{attribute 'linkalways'} 
{attribute 'no_explicit_call' := 'This FB is a CLASS and must be accessed using methods or properties'}
{attribute 'enable_dynamic_creation'}
FUNCTION_BLOCK Node_F_VN_HistogramExp EXTENDS VisionNode
VAR
	ipSrcImage : _ITcVnImage;
	ipMask : _ITcVnImage;
    ipDestHistogram : _ITcVnContainer;
	nBins : _UDINT(0);
	fLowerBound : _LREAL(0.0);
	fUpperBound : _LREAL(0.0);
    hrPrev : _HRESULT(S_OK);
	hresult : _HRESULT(S_OK);
END_VAR

METHOD PUBLIC  Clone : I_Node
VAR
	pNode : POINTER TO Node_F_VN_HistogramExp;
END_VAR
pNode := __NEW(Node_F_VN_HistogramExp);
Clone := pNode^;
END_METHOD

METHOD FB_init : BOOL
VAR_INPUT
	bInitRetains : BOOL; // if TRUE, the retain variables are initialized (warm start / cold start)
	bInCopyCode : BOOL;  // if TRUE, the instance afterwards gets moved into the copy code (online change)
END_VAR
AddInput('ipSrcImage', ipSrcImage);
AddInput('ipMask', ipMask);
AddInput('hrPrev', hrPrev);
AddParameter('nBins',nBins);
AddParameter('fLowerBound',fLowerBound);
AddParameter('fUpperBound',fUpperBound);
AddOutput('ipDestHistogram', ipDestHistogram);
AddOutput('hresult',hresult);
END_METHOD

METHOD PROTECTED OnExecute
hresult.Value := F_VN_HistogramExp(
	ipSrcImage := ipSrcImage.Value,
	ipDestHistogram := ipDestHistogram.Value,
	nBins := nBins.Value,
	fLowerBound := fLowerBound.Value,
	fUpperBound := fUpperBound.Value,
	ipMask := ipMask.Value,
	hrPrev := hrPrev.Value);
END_METHOD

METHOD PUBLIC PreExecutionCheck
VAR_INPUT
	Check : I_PreExecutionChecks;
END_VAR
Check.IsTrue(ipSrcImage.IsValid, 'ipSrcImage must contain an image');
END_METHOD

END_FUNCTION_BLOCK

(* stored: Version 1.1.0.1, ProductVersion 3.1.4026.18
   POU Node_F_VN_HistogramExp: Id {f5da5600-1207-0679-0d23-7a909a430501}, SpecialFunc None
   Folder Constructor: Id {ef3bb1f4-de02-043c-3d14-d546ae8a19af}
   Method Clone: Id {315b9e6d-9c21-0c08-079f-ff6853e39c95}
   Method FB_init: Id {2adac46d-5d71-03fb-36d0-0efd3f9dd5f5}
   Method OnExecute: Id {f9a155b1-b480-08fe-0246-3363c606746a}
   Method PreExecutionCheck: Id {fc254156-1d70-0042-1fb5-66a0d66495ac} *)
